Fanuc KAREL source: kd00005.KL

-- PROVISIONAL review KL for V1013-1; original PC SHA256 fcafbef2c10dd5457613fff9b04e9b40be86b6ed53dc3be2643cedff6618011e
-- Incomplete behavior may be omitted. Consult companion uncertainty JSON. Do not deploy.
PROGRAM KD00005
%NOLOCKGROUP
VAR
  I : INTEGER
  J : INTEGER
  B : BOOLEAN
  R : REAL
  S : STRING[80]
BEGIN
  -- UNRESOLVED_PC offsets 5-12; opcodes 9D,23
  -- UNRESOLVED_PC offsets 17-21; opcodes 7F
END KD00005
